// TIA Portal V19 export
FUNCTION "LAF_ControlEm" : Void   // FC15, LAD
TITLE = LAF_ControlEm
// This function provides the mode and state to the equipment module.
// stored: Access Published, SetENOAutomatically false
   VAR_INPUT
      isLinked : Bool;   // Information if EM is linked to Unit
   END_VAR
   VAR_OUTPUT
      unitStatusUsed : "LAF_typeUnitStatus";
   END_VAR
   VAR_IN_OUT
      unitStatus : "LAF_typeUnitStatus";
      hmiInterface : "LAF_typeEmInterface";   // HMI Manual commands
      localInterface : "LAF_typeEmControlNode";   // Local Manual commands
   END_VAR
   VAR_TEMP
      tempModeControlHmi : "LUC_typeModes";   // Temp of the HMI Manual Mode commands
      tempStateControlHmi : "LUC_typeStates";   // Temp of the HMI Manual State commands
      tempModePreviousCycle : "LUC_typeModes";   // Temp of the used Mode in the previous cycle
      tempStatusPreviousCycle : "LUC_typeStates";   // Temp of the used State in the previous cycle
   END_VAR
BEGIN

REGION Network 1: BLOCK INFO HEADER
   // Siemens AG / (c)Copyright 2024
   // -------------------------------------------------------------------------------
   // Title:            LAF_ControlEm
   // Comment/Function: This function provides the mode and state to the equipment module.
   // Library/Family:   LAF - Library of Automation Framework
   // Author:           Siemens Digital Industries
   // Tested with:      S7-PLCSIM Advanced V6.0 
   // Engineering:      TIA Portal V19
   // Restrictions:     -
   // Requirements:     -
   // -------------------------------------------------------------------------------
   // Change log table:
   // Version  | Date       | Expert in charge        | Changes applied
   // ----------|------------|-------------------------|-----------------------------
   // 01.01.00 | 21.06.2024 | SIMATIC Systems Support | First released version
   // 01.02.00 | 20.09.2024 | SIMATIC Systems Support | Block information properties updated and optimized code
END_REGION

REGION Network 2: DESCRIPTION
   // This block defines the modes and states for the equipment module.
   // If the EM is linked to the unit, the unit status is fully applied to the EM and a manual/direct EM control is not possible.
   // If the EM is not linked to the unit, the operator can set the mode and state manually, enable simulation and disable alarms. However, the Acknowledge commands and SafetyReleased are still taken from the unit.
   // Acknowledge and SafetyReleased from the unit are always applied, independently from being linked or not.
   // If controlled directly, the local interface has priority over the hmi interface
END_REGION

REGION Network 3 (SCL): Initialization
   // Read the HMI interface and map the HMI DWords to the Unit Structure and build temp Mode and State to be used
   #tempModeControlHmi.production := #hmiInterface.commands.directModeControl.%X0;
   #tempModeControlHmi.maintenance := #hmiInterface.commands.directModeControl.%X1;
   #tempModeControlHmi.manual := #hmiInterface.commands.directModeControl.%X2;
   #tempModeControlHmi.userMode01 := #hmiInterface.commands.directModeControl.%X3;
   #tempModeControlHmi.userMode02 := #hmiInterface.commands.directModeControl.%X4;
   #tempModeControlHmi.userMode03 := #hmiInterface.commands.directModeControl.%X5;
   #tempModeControlHmi.userMode04 := #hmiInterface.commands.directModeControl.%X6;
   #tempModeControlHmi.userMode05 := #hmiInterface.commands.directModeControl.%X7;
   #tempModeControlHmi.userMode06 := #hmiInterface.commands.directModeControl.%X8;
   #tempModeControlHmi.userMode07 := #hmiInterface.commands.directModeControl.%X9;
   #tempModeControlHmi.userMode08 := #hmiInterface.commands.directModeControl.%X10;
   #tempModeControlHmi.userMode09 := #hmiInterface.commands.directModeControl.%X11;
   #tempModeControlHmi.userMode10 := #hmiInterface.commands.directModeControl.%X12;
   #tempModeControlHmi.userMode11 := #hmiInterface.commands.directModeControl.%X13;
   #tempModeControlHmi.userMode12 := #hmiInterface.commands.directModeControl.%X14;
   #tempModeControlHmi.userMode13 := #hmiInterface.commands.directModeControl.%X15;

   #tempStateControlHmi.clearing := #hmiInterface.commands.directStateControl.%X0;
   #tempStateControlHmi.stopped := #hmiInterface.commands.directStateControl.%X1;
   #tempStateControlHmi.starting := #hmiInterface.commands.directStateControl.%X2;
   #tempStateControlHmi.idle := #hmiInterface.commands.directStateControl.%X3;
   #tempStateControlHmi.suspended := #hmiInterface.commands.directStateControl.%X4;
   #tempStateControlHmi.execute := #hmiInterface.commands.directStateControl.%X5;
   #tempStateControlHmi.stopping := #hmiInterface.commands.directStateControl.%X6;
   #tempStateControlHmi.aborting := #hmiInterface.commands.directStateControl.%X7;
   #tempStateControlHmi.aborted := #hmiInterface.commands.directStateControl.%X8;
   #tempStateControlHmi.holding := #hmiInterface.commands.directStateControl.%X9;
   #tempStateControlHmi.held := #hmiInterface.commands.directStateControl.%X10;
   #tempStateControlHmi.unholding := #hmiInterface.commands.directStateControl.%X11;
   #tempStateControlHmi.suspending := #hmiInterface.commands.directStateControl.%X12;
   #tempStateControlHmi.unsuspending := #hmiInterface.commands.directStateControl.%X13;
   #tempStateControlHmi.resetting := #hmiInterface.commands.directStateControl.%X14;
   #tempStateControlHmi.completing := #hmiInterface.commands.directStateControl.%X15;
   #tempStateControlHmi.complete := #hmiInterface.commands.directStateControl.%X16;

   // Last Cycle temp Mode and State to evaluate the new Mode and State
   #tempModePreviousCycle := #unitStatusUsed.mode;
   #tempStatusPreviousCycle := #unitStatusUsed.state;
END_REGION

REGION Network 4: Acknowledge
   // If EM is not linked, acknowledge from the unit are applied to the EM or can be controlled directly
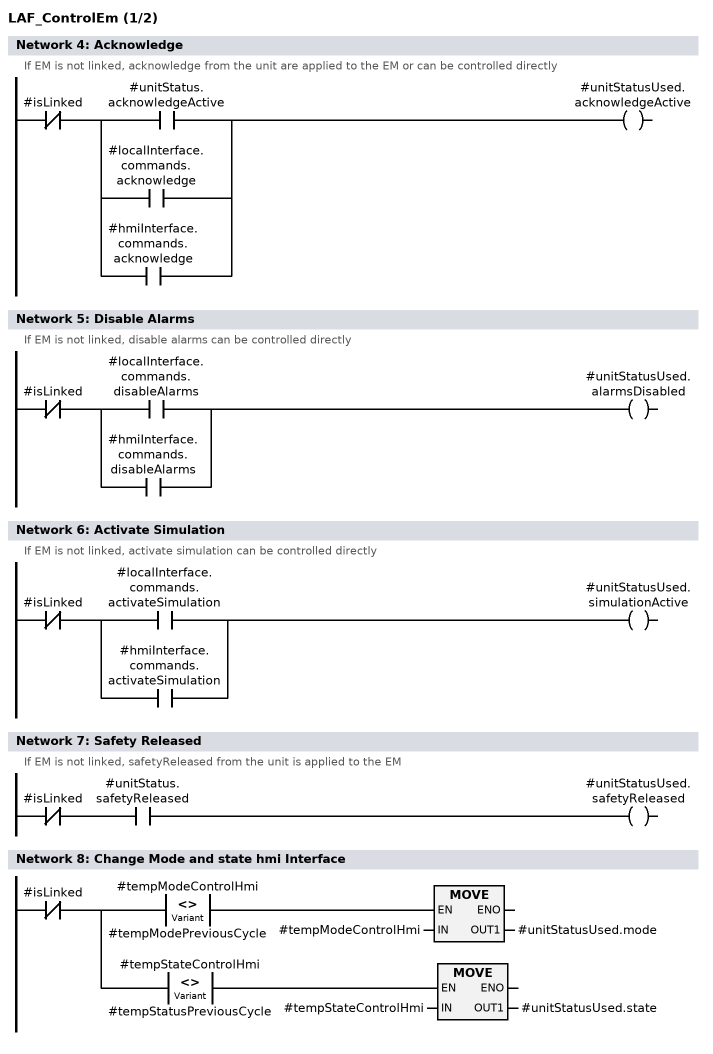
   RUNG wire#powerrail
      I_Contact( #isLinked )
      wire#w1
      Contact( #unitStatus.acknowledgeActive )
      wire#w2
      Coil( #unitStatusUsed.acknowledgeActive )
   END_RUNG
   RUNG wire#w1
      Contact( #localInterface.commands.acknowledge )
   END_RUNG wire#w2
   RUNG wire#w1
      Contact( #hmiInterface.commands.acknowledge )
   END_RUNG wire#w2
   // the same network as SCL:
   #unitStatusUsed.acknowledgeActive := NOT #isLinked AND (#unitStatus.acknowledgeActive OR #localInterface.commands.acknowledge OR #hmiInterface.commands.acknowledge);
END_REGION

REGION Network 5: Disable Alarms
   // If EM is not linked, disable alarms can be controlled directly
   RUNG wire#powerrail
      I_Contact( #isLinked )
      wire#w1
      Contact( #localInterface.commands.disableAlarms )
      wire#w2
      Coil( #unitStatusUsed.alarmsDisabled )
   END_RUNG
   RUNG wire#w1
      Contact( #hmiInterface.commands.disableAlarms )
   END_RUNG wire#w2
   // the same network as SCL:
   #unitStatusUsed.alarmsDisabled := NOT #isLinked AND (#localInterface.commands.disableAlarms OR #hmiInterface.commands.disableAlarms);
END_REGION

REGION Network 6: Activate Simulation
   // If EM is not linked, activate simulation can be controlled directly
   RUNG wire#powerrail
      I_Contact( #isLinked )
      wire#w1
      Contact( #localInterface.commands.activateSimulation )
      wire#w2
      Coil( #unitStatusUsed.simulationActive )
   END_RUNG
   RUNG wire#w1
      Contact( #hmiInterface.commands.activateSimulation )
   END_RUNG wire#w2
   // the same network as SCL:
   #unitStatusUsed.simulationActive := NOT #isLinked AND (#localInterface.commands.activateSimulation OR #hmiInterface.commands.activateSimulation);
END_REGION

REGION Network 7: Safety Released
   // If EM is not linked, safetyReleased from the unit is applied to the EM
   RUNG wire#powerrail
      I_Contact( #isLinked )
      Contact( #unitStatus.safetyReleased )
      Coil( #unitStatusUsed.safetyReleased )
   END_RUNG
   // the same network as SCL:
   #unitStatusUsed.safetyReleased := NOT #isLinked AND #unitStatus.safetyReleased;
END_REGION

REGION Network 8: Change Mode and state hmi Interface
   RUNG wire#powerrail
      I_Contact( #isLinked )
      wire#w1
      { S7_Templates := "SrcType := Variant" } NE_Contact(in1 := #tempModeControlHmi, in2 := #tempModePreviousCycle)
      Move(in := #tempModeControlHmi, out1 => #unitStatusUsed.mode)
   END_RUNG
   RUNG wire#w1
      { S7_Templates := "SrcType := Variant" } NE_Contact(in1 := #tempStateControlHmi, in2 := #tempStatusPreviousCycle)
      Move(in := #tempStateControlHmi, out1 => #unitStatusUsed.state)
   END_RUNG
   // the same network as SCL:
   IF NOT #isLinked AND (#tempModeControlHmi <> #tempModePreviousCycle) THEN
       #unitStatusUsed.mode := #tempModeControlHmi;
   END_IF;
   IF NOT #isLinked AND (#tempStateControlHmi <> #tempStatusPreviousCycle) THEN
       #unitStatusUsed.state := #tempStateControlHmi;
   END_IF;
END_REGION

REGION Network 9: Change Mode and state local Interface
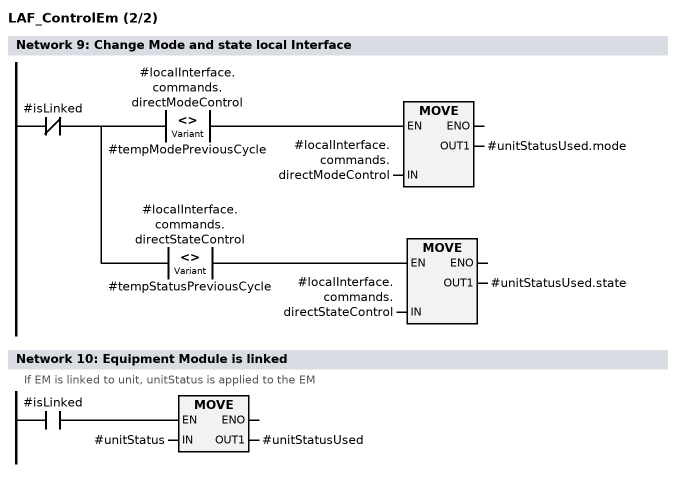
   RUNG wire#powerrail
      I_Contact( #isLinked )
      wire#w1
      { S7_Templates := "SrcType := Variant" } NE_Contact(in1 := #localInterface.commands.directModeControl, in2 := #tempModePreviousCycle)
      Move(in := #localInterface.commands.directModeControl, out1 => #unitStatusUsed.mode)
   END_RUNG
   RUNG wire#w1
      { S7_Templates := "SrcType := Variant" } NE_Contact(in1 := #localInterface.commands.directStateControl, in2 := #tempStatusPreviousCycle)
      Move(in := #localInterface.commands.directStateControl, out1 => #unitStatusUsed.state)
   END_RUNG
   // the same network as SCL:
   IF NOT #isLinked AND (#localInterface.commands.directModeControl <> #tempModePreviousCycle) THEN
       #unitStatusUsed.mode := #localInterface.commands.directModeControl;
   END_IF;
   IF NOT #isLinked AND (#localInterface.commands.directStateControl <> #tempStatusPreviousCycle) THEN
       #unitStatusUsed.state := #localInterface.commands.directStateControl;
   END_IF;
END_REGION

REGION Network 10: Equipment Module is linked
   // If EM is linked to unit, unitStatus is applied to the EM
   RUNG wire#powerrail
      Contact( #isLinked )
      Move(in := #unitStatus, out1 => #unitStatusUsed)
   END_RUNG
   // the same network as SCL:
   IF #isLinked THEN #unitStatusUsed := #unitStatus; END_IF;
END_REGION

REGION Network 11 (SCL): Update hmi and local interfaces
   // Update the internal unitStatusUsed variable to the hmi and local interfaces
   // Set the Interfaces to the new Mode & State
   #localInterface.commands.directModeControl := #tempModeControlHmi := #unitStatusUsed.mode;
   #localInterface.commands.directStateControl := #tempStateControlHmi := #unitStatusUsed.state;

   // Status bit update 
   #localInterface.status.acknowledgeActive := #unitStatusUsed.acknowledgeActive;
   #localInterface.status.alarmsDisabled := #unitStatusUsed.alarmsDisabled;
   #localInterface.status.safetyReleased := #unitStatusUsed.safetyReleased;
   #localInterface.status.simulationActive := #unitStatusUsed.simulationActive;

   // Transfer Status bits to the hmi status 
   #hmiInterface.status := #localInterface.status;
END_REGION

REGION Network 12 (SCL): Write Hmi Interface
   // Map the Unit Structure to the HMI DWords
   #hmiInterface.commands.directModeControl.%X0 := #tempModeControlHmi.production;
   #hmiInterface.commands.directModeControl.%X1 := #tempModeControlHmi.maintenance;
   #hmiInterface.commands.directModeControl.%X2 := #tempModeControlHmi.manual;
   #hmiInterface.commands.directModeControl.%X3 := #tempModeControlHmi.userMode01;
   #hmiInterface.commands.directModeControl.%X4 := #tempModeControlHmi.userMode02;
   #hmiInterface.commands.directModeControl.%X5 := #tempModeControlHmi.userMode03;
   #hmiInterface.commands.directModeControl.%X6 := #tempModeControlHmi.userMode04;
   #hmiInterface.commands.directModeControl.%X7 := #tempModeControlHmi.userMode05;
   #hmiInterface.commands.directModeControl.%X8 := #tempModeControlHmi.userMode06;
   #hmiInterface.commands.directModeControl.%X9 := #tempModeControlHmi.userMode07;
   #hmiInterface.commands.directModeControl.%X10 := #tempModeControlHmi.userMode08;
   #hmiInterface.commands.directModeControl.%X11 := #tempModeControlHmi.userMode09;
   #hmiInterface.commands.directModeControl.%X12 := #tempModeControlHmi.userMode10;
   #hmiInterface.commands.directModeControl.%X13 := #tempModeControlHmi.userMode11;
   #hmiInterface.commands.directModeControl.%X14 := #tempModeControlHmi.userMode12;
   #hmiInterface.commands.directModeControl.%X15 := #tempModeControlHmi.userMode13;

   #hmiInterface.commands.directStateControl.%X0 := #tempStateControlHmi.clearing;
   #hmiInterface.commands.directStateControl.%X1 := #tempStateControlHmi.stopped;
   #hmiInterface.commands.directStateControl.%X2 := #tempStateControlHmi.starting;
   #hmiInterface.commands.directStateControl.%X3 := #tempStateControlHmi.idle;
   #hmiInterface.commands.directStateControl.%X4 := #tempStateControlHmi.suspended;
   #hmiInterface.commands.directStateControl.%X5 := #tempStateControlHmi.execute;
   #hmiInterface.commands.directStateControl.%X6 := #tempStateControlHmi.stopping;
   #hmiInterface.commands.directStateControl.%X7 := #tempStateControlHmi.aborting;
   #hmiInterface.commands.directStateControl.%X8 := #tempStateControlHmi.aborted;
   #hmiInterface.commands.directStateControl.%X9 := #tempStateControlHmi.holding;
   #hmiInterface.commands.directStateControl.%X10 := #tempStateControlHmi.held;
   #hmiInterface.commands.directStateControl.%X11 := #tempStateControlHmi.unholding;
   #hmiInterface.commands.directStateControl.%X12 := #tempStateControlHmi.suspending;
   #hmiInterface.commands.directStateControl.%X13 := #tempStateControlHmi.unsuspending;
   #hmiInterface.commands.directStateControl.%X14 := #tempStateControlHmi.resetting;
   #hmiInterface.commands.directStateControl.%X15 := #tempStateControlHmi.completing;
   #hmiInterface.commands.directStateControl.%X16 := #tempStateControlHmi.complete;
END_REGION
END_FUNCTION
